{attribute 'pack_mode' := '0'}
TYPE ST_FurnaceOut :
STRUCT
	bPWMSignal					: BOOL;
END_STRUCT
END_TYPE

(* stored: Version 1.1.0.1
   DUT ST_FurnaceOut: Id {8e06e916-a8ac-4787-9d35-a05c91a5faf9} *)
